FUNCTION_BLOCK ZAppSequenceRunning EXTENDS ZAppSequence IMPLEMENTS ZCore.ISequence
VAR
  _step : ZCore.Step(ZAppStep.RunningBegin, ZAppStep.RunningEnd);
END_VAR

IF OnStart(_step)
THEN
  // init custom sequence variables here ...
END_IF

REPEAT
  LogStep();

  CASE _step.Index OF
    (* -------------------------------------------------------------------------------------------------------------------------------- *)
    ZAppStep.RunningBegin:
    (* -------------------------------------------------------------------------------------------------------------------------------- *)
      ; // implement me
      
    (* -------------------------------------------------------------------------------------------------------------------------------- *)
    ZAppStep.RunningEnd:
    (* -------------------------------------------------------------------------------------------------------------------------------- *)
      SetBusy(FALSE);
      
  ELSE
    Abort('sequence contains unhandled step');
  END_CASE
UNTIL _step.IsNotRepeatable() OR_ELSE NOT Busy END_REPEAT

END_FUNCTION_BLOCK

(* stored: Version 1.1.0.1
   POU ZAppSequenceRunning: Id {af7b56e7-20f5-4294-ac1e-f2e4bdce2b8b}, SpecialFunc None *)
